FUNCTION_BLOCK FB_A
VAR_INPUT
    nVarA: INT;
END_VAR

nVarA := 1;

END_FUNCTION_BLOCK

(* stored: Version 1.1.0.1, ProductVersion 3.1.4024.12
   POU FB_A: Id {09e457a3-e2f8-4454-833e-cb8ce6430a0c}, SpecialFunc None *)
